FUNCTION_BLOCK FB_HMI_COMPONENT
VAR_INPUT
END_VAR
VAR_OUTPUT
    fbHealthStatus : FB_HMI_HEALTH_STATUS;
    fbBusyStatus : FB_HMI_BUSY_STATUS;
    fbStatusColor : T_HMI_COLORS;
END_VAR
VAR
END_VAR

METHOD PROTECTED M_UpdateStatusColor
VAR_INPUT
END_VAR
// health and busy states must be updated by the subtype before calling this method!
fbStatusColor := F_HMI_HEALTH_BUSY_TO_COLOR(fbHealthStatus, fbBusyStatus);
END_METHOD

END_FUNCTION_BLOCK

(* stored: Version 1.1.0.1, ProductVersion 3.1.4024.14
   POU FB_HMI_COMPONENT: Id {7c0d017e-864e-4210-8c94-e5ade760e15b}, SpecialFunc None
   Method M_UpdateStatusColor: Id {d83e0729-6281-4c94-b757-bf3e108374e5} *)
